Yaskawa INFORM job: HOME.JBI

/JOB
//NAME HOME
//POS
///NPOS 1,1,1,0,0,0
///TOOL 2
///POSTYPE PULSE
///PULSE
C00000=0,0,0,0,0,0
///TOOL 0
BC00000=0
EC00000=0,0
//INST
///DATE 2026/05/13 10:02
///ATTR SC,RW
///GROUP1 RB1,BS1
///GROUP2 ST1
NOP
'Home
MEMOF
CLEAR MPF
MOVJ C00000 BC00000 VJ=100.00  +MOVJ EC00000 VJ=100.00
END
